TYPE commSignal :
STRUCT
	address : WORD;	//0
	widthOn : WORD; //1
	widthOff : WORD; //2
	widthOnCount : WORD;//3
	widthOffCount : WORD;//4
	outputWord: WORD;//5
END_STRUCT
END_TYPE

(* stored: Version 1.1.0.1, ProductVersion 3.1.4022.10
   DUT commSignal: Id {bdbdac30-612d-430e-bbcf-43f1cafaa021} *)
